// TIA Portal V15.1 export
// export: Created 2020-12-11T18:23:40.5486827Z, ExportSetting WithDefaults, WithReadOnly, DisplayName Totally Integrated Automation Portal, DisplayVersion V15.1 Update 4, DisplayName TIA Portal Openness, DisplayVersion V15.1, DisplayName SINAMICS Startdrive Advanced, DisplayVersion V15.1 Update3, DisplayName SINAMICS Startdrive G110M, G120, G120C, G120D, G120P, DisplayVersion V15.1 Update3, DisplayName SINAMICS Startdrive G130, G150, S120, S150, SINAMICS MV, S210, DisplayVersion V15.1 Update3, DisplayName STEP 7 Professional, DisplayVersion V15.1 Update 4, DisplayName STEP 7 Safety, DisplayVersion V15.1, DisplayName WinCC Professional, DisplayVersion V15.1 Update 4
PlcWatchTable "IO_ST_A"
  PlcTableCommentEntry   Comment="D1"
  PlcWatchTableEntry "Hello world"  Address=%I2001.0, DisplayFormat=Bool, ModifyTrigger=Permanent, MonitorTrigger=Permanent
  PlcWatchTableEntry ""SQ86/BA""  Address=%I2000.1, DisplayFormat=Bool, ModifyTrigger=Permanent, MonitorTrigger=Permanent
  PlcWatchTableEntry ""SQ87/BA""  Address=%I2001.1, DisplayFormat=Bool, ModifyTrigger=Permanent, MonitorTrigger=Permanent
  PlcWatchTableEntry ""SQ57/BA""  Address=%I2000.2, DisplayFormat=Bool, ModifyTrigger=Permanent, MonitorTrigger=Permanent
  PlcWatchTableEntry ""SQ58/BA""  Address=%I2001.2, DisplayFormat=Bool, ModifyTrigger=Permanent, MonitorTrigger=Permanent
  PlcWatchTableEntry ""SQ59/BA""  Address=%I2000.3, DisplayFormat=Bool, ModifyTrigger=Permanent, MonitorTrigger=Permanent
  PlcWatchTableEntry ""SQ60/BA""  Address=%I2001.3, DisplayFormat=Bool, ModifyTrigger=Permanent, MonitorTrigger=Permanent
  PlcWatchTableEntry ""SQ73/BA""  Address=%I2000.4, DisplayFormat=Bool, ModifyTrigger=Permanent, MonitorTrigger=Permanent
  PlcWatchTableEntry ""SQ74/BA""  Address=%I2001.4, DisplayFormat=Bool, ModifyTrigger=Permanent, MonitorTrigger=Permanent
  PlcWatchTableEntry ""SQ31/BA""  Address=%I2000.5, DisplayFormat=Bool, ModifyTrigger=Permanent, MonitorTrigger=Permanent
  PlcWatchTableEntry ""SQ32/BA""  Address=%I2001.5, DisplayFormat=Bool, ModifyTrigger=Permanent, MonitorTrigger=Permanent
  PlcWatchTableEntry ""FTC2/BA""  Address=%I2000.6, DisplayFormat=Bool, ModifyTrigger=Permanent, MonitorTrigger=Permanent
  PlcWatchTableEntry ""SQ15/BA""  Address=%I2001.6, DisplayFormat=Bool, ModifyTrigger=Permanent, MonitorTrigger=Permanent
  PlcWatchTableEntry ""FTC1/BA""  Address=%I2000.7, DisplayFormat=Bool, ModifyTrigger=Permanent, MonitorTrigger=Permanent
  PlcWatchTableEntry ""FTC3/BA""  Address=%I2001.7, DisplayFormat=Bool, ModifyTrigger=Permanent, MonitorTrigger=Permanent
  PlcTableCommentEntry   Comment="D2"
  PlcWatchTableEntry ""SQ61/BA""  Address=%I2002.0, DisplayFormat=Bool, ModifyTrigger=Permanent, MonitorTrigger=Permanent
  PlcWatchTableEntry ""SQ62/BA""  Address=%I2003.0, DisplayFormat=Bool, ModifyTrigger=Permanent, MonitorTrigger=Permanent
  PlcWatchTableEntry ""SQ66/BA""  Address=%I2002.1, DisplayFormat=Bool, ModifyTrigger=Permanent, MonitorTrigger=Permanent
  PlcWatchTableEntry ""SQ67/BA""  Address=%I2003.1, DisplayFormat=Bool, ModifyTrigger=Permanent, MonitorTrigger=Permanent
  PlcWatchTableEntry ""SQ68/BA""  Address=%I2002.2, DisplayFormat=Bool, ModifyTrigger=Permanent, MonitorTrigger=Permanent
  PlcWatchTableEntry ""SQ72/BA""  Address=%I2003.2, DisplayFormat=Bool, ModifyTrigger=Permanent, MonitorTrigger=Permanent
  PlcWatchTableEntry ""SQ8/BA""  Address=%I2002.3, DisplayFormat=Bool, ModifyTrigger=Permanent, MonitorTrigger=Permanent
  PlcWatchTableEntry ""SQ9/BA""  Address=%I2003.3, DisplayFormat=Bool, ModifyTrigger=Permanent, MonitorTrigger=Permanent
  PlcWatchTableEntry ""SQ80/BA""  Address=%I2002.4, DisplayFormat=Bool, ModifyTrigger=Permanent, MonitorTrigger=Permanent
  PlcWatchTableEntry ""SQ81/BA""  Address=%I2003.4, DisplayFormat=Bool, ModifyTrigger=Permanent, MonitorTrigger=Permanent
  PlcWatchTableEntry ""FTC15/BA""  Address=%I2002.5, DisplayFormat=Bool, ModifyTrigger=Permanent, MonitorTrigger=Permanent
  PlcWatchTableEntry ""FTC92/BA""  Address=%I2003.5, DisplayFormat=Bool, ModifyTrigger=Permanent, MonitorTrigger=Permanent
  PlcWatchTableEntry ""FTC93/BA""  Address=%I2002.6, DisplayFormat=Bool, ModifyTrigger=Permanent, MonitorTrigger=Permanent
  PlcWatchTableEntry ""FTC94/BA""  Address=%I2003.6, DisplayFormat=Bool, ModifyTrigger=Permanent, MonitorTrigger=Permanent
  PlcWatchTableEntry ""SQ_SPARE_31/BA""  Address=%I2002.7, DisplayFormat=Bool, ModifyTrigger=Permanent, MonitorTrigger=Permanent
  PlcWatchTableEntry ""SQ_SPARE_32/BA""  Address=%I2003.7, DisplayFormat=Bool, ModifyTrigger=Permanent, MonitorTrigger=Permanent
  PlcTableCommentEntry   Comment="D3 - REMOVED"
  PlcWatchTableEntry ""SQ_SPARE_33/BA""  Address=%I2004.0, DisplayFormat=Bool, ModifyTrigger=Permanent, MonitorTrigger=Permanent
  PlcWatchTableEntry ""SQ_SPARE_34/BA""  Address=%I2005.0, DisplayFormat=Bool, ModifyTrigger=Permanent, MonitorTrigger=Permanent
  PlcWatchTableEntry ""SQ_SPARE_35/BA""  Address=%I2004.1, DisplayFormat=Bool, ModifyTrigger=Permanent, MonitorTrigger=Permanent
  PlcWatchTableEntry ""SQ_SPARE_36/BA""  Address=%I2005.1, DisplayFormat=Bool, ModifyTrigger=Permanent, MonitorTrigger=Permanent
  PlcWatchTableEntry ""SQ_SPARE_37/BA""  Address=%I2004.2, DisplayFormat=Bool, ModifyTrigger=Permanent, MonitorTrigger=Permanent
  PlcWatchTableEntry ""SQ_SPARE_38/BA""  Address=%I2005.2, DisplayFormat=Bool, ModifyTrigger=Permanent, MonitorTrigger=Permanent
  PlcWatchTableEntry ""SQ_SPARE_39/BA""  Address=%I2004.3, DisplayFormat=Bool, ModifyTrigger=Permanent, MonitorTrigger=Permanent
  PlcWatchTableEntry ""SQ_SPARE_40/BA""  Address=%I2005.3, DisplayFormat=Bool, ModifyTrigger=Permanent, MonitorTrigger=Permanent
  PlcWatchTableEntry ""SQ_SPARE_41/BA""  Address=%I2004.4, DisplayFormat=Bool, ModifyTrigger=Permanent, MonitorTrigger=Permanent
  PlcWatchTableEntry ""SQ_SPARE_42/BA""  Address=%I2005.4, DisplayFormat=Bool, ModifyTrigger=Permanent, MonitorTrigger=Permanent
  PlcWatchTableEntry ""SQ_SPARE_43/BA""  Address=%I2004.5, DisplayFormat=Bool, ModifyTrigger=Permanent, MonitorTrigger=Permanent
  PlcWatchTableEntry ""SQ_SPARE_44/BA""  Address=%I2005.5, DisplayFormat=Bool, ModifyTrigger=Permanent, MonitorTrigger=Permanent
  PlcWatchTableEntry ""SQ_SPARE_45/BA""  Address=%I2004.6, DisplayFormat=Bool, ModifyTrigger=Permanent, MonitorTrigger=Permanent
  PlcWatchTableEntry ""SQ_SPARE_46/BA""  Address=%I2005.6, DisplayFormat=Bool, ModifyTrigger=Permanent, MonitorTrigger=Permanent
  PlcWatchTableEntry ""SQ_SPARE_47/BA""  Address=%I2004.7, DisplayFormat=Bool, ModifyTrigger=Permanent, MonitorTrigger=Permanent
  PlcWatchTableEntry ""SQ_SPARE_48/BA""  Address=%I2005.7, DisplayFormat=Bool, ModifyTrigger=Permanent, MonitorTrigger=Permanent
  PlcTableCommentEntry   Comment="D2A"
  PlcWatchTableEntry ""FTC5/BA""  Address=%I2006.0, DisplayFormat=Bool, ModifyTrigger=Permanent, MonitorTrigger=Permanent
  PlcWatchTableEntry ""FTC6/BA""  Address=%I2007.0, DisplayFormat=Bool, ModifyTrigger=Permanent, MonitorTrigger=Permanent
  PlcWatchTableEntry ""FTC7/BA""  Address=%I2006.1, DisplayFormat=Bool, ModifyTrigger=Permanent, MonitorTrigger=Permanent
  PlcWatchTableEntry ""SQ95/BA""  Address=%I2007.1, DisplayFormat=Bool, ModifyTrigger=Permanent, MonitorTrigger=Permanent
  PlcWatchTableEntry ""SQ_SPARE_99/BA""  Address=%I2006.2, DisplayFormat=Bool, ModifyTrigger=Permanent, MonitorTrigger=Permanent
  PlcWatchTableEntry ""SQ_SPARE_107/BA""  Address=%I2007.2, DisplayFormat=Bool, ModifyTrigger=Permanent, MonitorTrigger=Permanent
  PlcWatchTableEntry ""FTC90/BA""  Address=%I2006.3, DisplayFormat=Bool, ModifyTrigger=Permanent, MonitorTrigger=Permanent
  PlcWatchTableEntry ""SQ96/BA""  Address=%I2007.3, DisplayFormat=Bool, ModifyTrigger=Permanent, MonitorTrigger=Permanent
  PlcWatchTableEntry ""SQ_SPARE_101/BA""  Address=%I2006.4, DisplayFormat=Bool, ModifyTrigger=Permanent, MonitorTrigger=Permanent
  PlcWatchTableEntry ""SQ_SPARE_109/BA""  Address=%I2007.4, DisplayFormat=Bool, ModifyTrigger=Permanent, MonitorTrigger=Permanent
  PlcWatchTableEntry ""SQ_SPARE_102/BA""  Address=%I2006.5, DisplayFormat=Bool, ModifyTrigger=Permanent, MonitorTrigger=Permanent
  PlcWatchTableEntry ""SQ_SPARE_110/BA""  Address=%I2007.5, DisplayFormat=Bool, ModifyTrigger=Permanent, MonitorTrigger=Permanent
  PlcWatchTableEntry ""SQ_SPARE_103/BA""  Address=%I2006.6, DisplayFormat=Bool, ModifyTrigger=Permanent, MonitorTrigger=Permanent
  PlcWatchTableEntry ""SQ_SPARE_111/BA""  Address=%I2007.6, DisplayFormat=Bool, ModifyTrigger=Permanent, MonitorTrigger=Permanent
  PlcWatchTableEntry ""SQ_SPARE_104/BA""  Address=%I2006.7, DisplayFormat=Bool, ModifyTrigger=Permanent, MonitorTrigger=Permanent
  PlcWatchTableEntry ""SQ_SPARE_112/BA""  Address=%I2007.7, DisplayFormat=Bool, ModifyTrigger=Permanent, MonitorTrigger=Permanent
  PlcTableCommentEntry   Comment="D4"
  PlcWatchTableEntry ""SQ44/BA""  Address=%I2100.0, DisplayFormat=Bool, ModifyTrigger=Permanent, MonitorTrigger=Permanent
  PlcWatchTableEntry ""SQ45/BA""  Address=%I2101.0, DisplayFormat=Bool, ModifyTrigger=Permanent, MonitorTrigger=Permanent
  PlcWatchTableEntry ""SQ89/BA""  Address=%I2101.1, DisplayFormat=Bool, ModifyTrigger=Permanent, MonitorTrigger=Permanent
  PlcWatchTableEntry ""SQ88/BA""  Address=%I2100.1, DisplayFormat=Bool, ModifyTrigger=Permanent, MonitorTrigger=Permanent
  PlcWatchTableEntry ""SQ48/BA""  Address=%I2100.2, DisplayFormat=Bool, ModifyTrigger=Permanent, MonitorTrigger=Permanent
  PlcWatchTableEntry ""SQ49/BA""  Address=%I2101.2, DisplayFormat=Bool, ModifyTrigger=Permanent, MonitorTrigger=Permanent
  PlcWatchTableEntry ""SQ50/BA""  Address=%I2100.3, DisplayFormat=Bool, ModifyTrigger=Permanent, MonitorTrigger=Permanent
  PlcWatchTableEntry ""SQ51/BA""  Address=%I2101.3, DisplayFormat=Bool, ModifyTrigger=Permanent, MonitorTrigger=Permanent
  PlcWatchTableEntry ""SQ75/BA""  Address=%I2100.4, DisplayFormat=Bool, ModifyTrigger=Permanent, MonitorTrigger=Permanent
  PlcWatchTableEntry ""SQ76/BA""  Address=%I2101.4, DisplayFormat=Bool, ModifyTrigger=Permanent, MonitorTrigger=Permanent
  PlcWatchTableEntry ""SQ18/BA""  Address=%I2100.5, DisplayFormat=Bool, ModifyTrigger=Permanent, MonitorTrigger=Permanent
  PlcWatchTableEntry ""SQ19/BA""  Address=%I2101.5, DisplayFormat=Bool, ModifyTrigger=Permanent, MonitorTrigger=Permanent
  PlcWatchTableEntry ""SQ97/BA""  Address=%I2100.6, DisplayFormat=Bool, ModifyTrigger=Permanent, MonitorTrigger=Permanent
  PlcWatchTableEntry ""SQ17/BA""  Address=%I2101.6, DisplayFormat=Bool, ModifyTrigger=Permanent, MonitorTrigger=Permanent
  PlcWatchTableEntry ""SQ98/BA""  Address=%I2100.7, DisplayFormat=Bool, ModifyTrigger=Permanent, MonitorTrigger=Permanent
  PlcWatchTableEntry ""SQ_SPARE_64/BA""  Address=%I2101.7, DisplayFormat=Bool, ModifyTrigger=Permanent, MonitorTrigger=Permanent
  PlcTableCommentEntry   Comment="D5 - REMOVED"
  PlcWatchTableEntry ""SQ_SPARE_65/BA""  Address=%I2102.0, DisplayFormat=Bool, ModifyTrigger=Permanent, MonitorTrigger=Permanent
  PlcWatchTableEntry ""SQ_SPARE_66/BA""  Address=%I2103.0, DisplayFormat=Bool, ModifyTrigger=Permanent, MonitorTrigger=Permanent
  PlcWatchTableEntry ""SQ_SPARE_67/BA""  Address=%I2102.1, DisplayFormat=Bool, ModifyTrigger=Permanent, MonitorTrigger=Permanent
  PlcWatchTableEntry ""SQ_SPARE_68/BA""  Address=%I2103.1, DisplayFormat=Bool, ModifyTrigger=Permanent, MonitorTrigger=Permanent
  PlcWatchTableEntry ""SQ_SPARE_69/BA""  Address=%I2102.2, DisplayFormat=Bool, ModifyTrigger=Permanent, MonitorTrigger=Permanent
  PlcWatchTableEntry ""SQ_SPARE_70/BA""  Address=%I2103.2, DisplayFormat=Bool, ModifyTrigger=Permanent, MonitorTrigger=Permanent
  PlcWatchTableEntry ""SQ_SPARE_71/BA""  Address=%I2102.3, DisplayFormat=Bool, ModifyTrigger=Permanent, MonitorTrigger=Permanent
  PlcWatchTableEntry ""SQ_SPARE_72/BA""  Address=%I2103.3, DisplayFormat=Bool, ModifyTrigger=Permanent, MonitorTrigger=Permanent
  PlcWatchTableEntry ""SQ_SPARE_73/BA""  Address=%I2102.4, DisplayFormat=Bool, ModifyTrigger=Permanent, MonitorTrigger=Permanent
  PlcWatchTableEntry ""SQ_SPARE_74/BA""  Address=%I2103.4, DisplayFormat=Bool, ModifyTrigger=Permanent, MonitorTrigger=Permanent
  PlcWatchTableEntry ""SQ_SPARE_75/BA""  Address=%I2102.5, DisplayFormat=Bool, ModifyTrigger=Permanent, MonitorTrigger=Permanent
  PlcWatchTableEntry ""SQ_SPARE_76/BA""  Address=%I2103.5, DisplayFormat=Bool, ModifyTrigger=Permanent, MonitorTrigger=Permanent
  PlcWatchTableEntry ""SQ_SPARE_77/BA""  Address=%I2102.6, DisplayFormat=Bool, ModifyTrigger=Permanent, MonitorTrigger=Permanent
  PlcWatchTableEntry ""SQ_SPARE_78/BA""  Address=%I2103.6, DisplayFormat=Bool, ModifyTrigger=Permanent, MonitorTrigger=Permanent
  PlcWatchTableEntry ""SQ_SPARE_79/BA""  Address=%I2102.7, DisplayFormat=Bool, ModifyTrigger=Permanent, MonitorTrigger=Permanent
  PlcWatchTableEntry ""SQ_SPARE_80/BA""  Address=%I2103.7, DisplayFormat=Bool, ModifyTrigger=Permanent, MonitorTrigger=Permanent
  PlcTableCommentEntry   Comment="D6"
  PlcWatchTableEntry ""SQ69/BA""  Address=%I2104.0, DisplayFormat=Bool, ModifyTrigger=Permanent, MonitorTrigger=Permanent
  PlcWatchTableEntry ""SQ70/BA""  Address=%I2105.0, DisplayFormat=Bool, ModifyTrigger=Permanent, MonitorTrigger=Permanent
  PlcWatchTableEntry ""SQ71/BA""  Address=%I2104.1, DisplayFormat=Bool, ModifyTrigger=Permanent, MonitorTrigger=Permanent
  PlcWatchTableEntry ""SQ77/BA""  Address=%I2105.1, DisplayFormat=Bool, ModifyTrigger=Permanent, MonitorTrigger=Permanent
  PlcWatchTableEntry ""SQ78/BA""  Address=%I2104.2, DisplayFormat=Bool, ModifyTrigger=Permanent, MonitorTrigger=Permanent
  PlcWatchTableEntry ""SQ79/BA""  Address=%I2105.2, DisplayFormat=Bool, ModifyTrigger=Permanent, MonitorTrigger=Permanent
  PlcWatchTableEntry ""SQ6/BA""  Address=%I2104.3, DisplayFormat=Bool, ModifyTrigger=Permanent, MonitorTrigger=Permanent
  PlcWatchTableEntry ""SQ7/BA""  Address=%I2105.3, DisplayFormat=Bool, ModifyTrigger=Permanent, MonitorTrigger=Permanent
  PlcWatchTableEntry ""SQ82/BA""  Address=%I2104.4, DisplayFormat=Bool, ModifyTrigger=Permanent, MonitorTrigger=Permanent
  PlcWatchTableEntry ""SQ83/BA""  Address=%I2105.4, DisplayFormat=Bool, ModifyTrigger=Permanent, MonitorTrigger=Permanent
  PlcWatchTableEntry ""SQ_SPARE_91/BA""  Address=%I2104.5, DisplayFormat=Bool, ModifyTrigger=Permanent, MonitorTrigger=Permanent
  PlcWatchTableEntry ""SQ_SPARE_92/BA""  Address=%I2105.5, DisplayFormat=Bool, ModifyTrigger=Permanent, MonitorTrigger=Permanent
  PlcWatchTableEntry ""SQ_SPARE_93/BA""  Address=%I2104.6, DisplayFormat=Bool, ModifyTrigger=Permanent, MonitorTrigger=Permanent
  PlcWatchTableEntry ""SQ_SPARE_94/BA""  Address=%I2105.6, DisplayFormat=Bool, ModifyTrigger=Permanent, MonitorTrigger=Permanent
  PlcWatchTableEntry ""SQ_SPARE_95/BA""  Address=%I2104.7, DisplayFormat=Bool, ModifyTrigger=Permanent, MonitorTrigger=Permanent
  PlcWatchTableEntry ""SQ_SPARE_96/BA""  Address=%I2105.7, DisplayFormat=Bool, ModifyTrigger=Permanent, MonitorTrigger=Permanent
  PlcTableCommentEntry   Comment="D6A"
  PlcWatchTableEntry ""SQ_SPARE_113/BA""  Address=%I2106.0, DisplayFormat=Bool, ModifyTrigger=Permanent, MonitorTrigger=Permanent
  PlcWatchTableEntry ""SQ_SPARE_114/BA""  Address=%I2106.1, DisplayFormat=Bool, ModifyTrigger=Permanent, MonitorTrigger=Permanent
  PlcWatchTableEntry ""SQ_SPARE_115/BA""  Address=%I2106.2, DisplayFormat=Bool, ModifyTrigger=Permanent, MonitorTrigger=Permanent
  PlcWatchTableEntry ""SQ_SPARE_116/BA""  Address=%I2106.3, DisplayFormat=Bool, ModifyTrigger=Permanent, MonitorTrigger=Permanent
  PlcWatchTableEntry ""FTC91/BA""  Address=%I2106.4, DisplayFormat=Bool, ModifyTrigger=Permanent, MonitorTrigger=Permanent
  PlcWatchTableEntry ""SQ_SPARE_118/BA""  Address=%I2106.5, DisplayFormat=Bool, ModifyTrigger=Permanent, MonitorTrigger=Permanent
  PlcWatchTableEntry ""SQ_SPARE_119/BA""  Address=%I2106.6, DisplayFormat=Bool, ModifyTrigger=Permanent, MonitorTrigger=Permanent
  PlcWatchTableEntry ""SQ_SPARE_120/BA""  Address=%I2106.7, DisplayFormat=Bool, ModifyTrigger=Permanent, MonitorTrigger=Permanent
  PlcWatchTableEntry ""SQ_SPARE_121/BA""  Address=%I2107.0, DisplayFormat=Bool, ModifyTrigger=Permanent, MonitorTrigger=Permanent
  PlcWatchTableEntry ""SQ_SPARE_122/BA""  Address=%I2107.1, DisplayFormat=Bool, ModifyTrigger=Permanent, MonitorTrigger=Permanent
  PlcWatchTableEntry ""SQ_SPARE_123/BA""  Address=%I2107.2, DisplayFormat=Bool, ModifyTrigger=Permanent, MonitorTrigger=Permanent
  PlcWatchTableEntry ""SQ_SPARE_124/BA""  Address=%I2107.3, DisplayFormat=Bool, ModifyTrigger=Permanent, MonitorTrigger=Permanent
  PlcWatchTableEntry ""SQ_SPARE_125/BA""  Address=%I2107.4, DisplayFormat=Bool, ModifyTrigger=Permanent, MonitorTrigger=Permanent
  PlcWatchTableEntry ""SQ_SPARE_126/BA""  Address=%I2107.5, DisplayFormat=Bool, ModifyTrigger=Permanent, MonitorTrigger=Permanent
  PlcWatchTableEntry ""SQ_SPARE_127/BA""  Address=%I2107.6, DisplayFormat=Bool, ModifyTrigger=Permanent, MonitorTrigger=Permanent
  PlcWatchTableEntry ""SQ_SPARE_128/BA""  Address=%I2107.7, DisplayFormat=Bool, ModifyTrigger=Permanent, MonitorTrigger=Permanent
  PlcWatchTableEntry   DisplayFormat=Undef, ModifyTrigger=Undef, MonitorTrigger=Undef
  PlcWatchTableEntry   DisplayFormat=Undef, ModifyTrigger=Undef, MonitorTrigger=Undef
  PlcWatchTableEntry   DisplayFormat=Undef, ModifyTrigger=Undef, MonitorTrigger=Undef
  PlcWatchTableEntry   DisplayFormat=Undef, ModifyTrigger=Undef, MonitorTrigger=Undef
  PlcWatchTableEntry   Address=%QB0, DisplayFormat=Hex, ModifyTrigger=Permanent, ModifyValue=16#FF, MonitorTrigger=Permanent
  PlcWatchTableEntry ""Y1A/BA""  Address=%Q2000.0, DisplayFormat=Bool, ModifyTrigger=Permanent, MonitorTrigger=Permanent
  PlcWatchTableEntry ""Y1B/BA""  Address=%Q2000.1, DisplayFormat=Bool, ModifyTrigger=Permanent, MonitorTrigger=Permanent
  PlcWatchTableEntry ""Y2A/BA""  Address=%Q2000.2, DisplayFormat=Bool, ModifyTrigger=Permanent, MonitorTrigger=Permanent
  PlcWatchTableEntry ""Y2B/BA""  Address=%Q2000.3, DisplayFormat=Bool, ModifyTrigger=Permanent, MonitorTrigger=Permanent
  PlcWatchTableEntry ""Y3A/BA""  Address=%Q2000.4, DisplayFormat=Bool, ModifyTrigger=Permanent, MonitorTrigger=Permanent
  PlcWatchTableEntry ""Y3B/BA""  Address=%Q2000.5, DisplayFormat=Bool, ModifyTrigger=Permanent, MonitorTrigger=Permanent
  PlcWatchTableEntry ""Y4A/BA""  Address=%Q2000.6, DisplayFormat=Bool, ModifyTrigger=Permanent, MonitorTrigger=Permanent
  PlcWatchTableEntry ""Y4B/BA""  Address=%Q2000.7, DisplayFormat=Bool, ModifyTrigger=Permanent, MonitorTrigger=Permanent
  PlcWatchTableEntry ""Y5A/BA""  Address=%Q2001.0, DisplayFormat=Bool, ModifyTrigger=Permanent, MonitorTrigger=Permanent
  PlcWatchTableEntry ""Y5B/BA""  Address=%Q2001.1, DisplayFormat=Bool, ModifyTrigger=Permanent, MonitorTrigger=Permanent
  PlcWatchTableEntry ""Y6A/BA""  Address=%Q2001.2, DisplayFormat=Bool, ModifyTrigger=Permanent, MonitorTrigger=Permanent
  PlcWatchTableEntry ""Y6B/BA""  Address=%Q2001.3, DisplayFormat=Bool, ModifyTrigger=Permanent, MonitorTrigger=Permanent
  PlcWatchTableEntry ""Y7A/BA""  Address=%Q2001.4, DisplayFormat=Bool, ModifyTrigger=Permanent, MonitorTrigger=Permanent
  PlcWatchTableEntry ""Y7B/BA""  Address=%Q2001.5, DisplayFormat=Bool, ModifyTrigger=Permanent, MonitorTrigger=Permanent
  PlcWatchTableEntry ""Y8A/BA""  Address=%Q2001.6, DisplayFormat=Bool, ModifyTrigger=Permanent, MonitorTrigger=Permanent
  PlcWatchTableEntry ""Y8B/BA""  Address=%Q2001.7, DisplayFormat=Bool, ModifyTrigger=Permanent, MonitorTrigger=Permanent
  PlcWatchTableEntry ""Y9A/BA""  Address=%Q2002.0, DisplayFormat=Bool, ModifyTrigger=Permanent, MonitorTrigger=Permanent
  PlcWatchTableEntry ""Y9B/BA""  Address=%Q2002.1, DisplayFormat=Bool, ModifyTrigger=Permanent, MonitorTrigger=Permanent
  PlcWatchTableEntry ""Y10A/BA""  Address=%Q2002.2, DisplayFormat=Bool, ModifyTrigger=Permanent, MonitorTrigger=Permanent
  PlcWatchTableEntry ""Y10B/BA""  Address=%Q2002.3, DisplayFormat=Bool, ModifyTrigger=Permanent, MonitorTrigger=Permanent
  PlcWatchTableEntry ""Y11A/BA""  Address=%Q2002.4, DisplayFormat=Bool, ModifyTrigger=Permanent, MonitorTrigger=Permanent
  PlcWatchTableEntry ""Y11B/BA""  Address=%Q2002.5, DisplayFormat=Bool, ModifyTrigger=Permanent, MonitorTrigger=Permanent
  PlcWatchTableEntry ""Y12A/BA""  Address=%Q2002.6, DisplayFormat=Bool, ModifyTrigger=Permanent, MonitorTrigger=Permanent
  PlcWatchTableEntry ""Y12B/BA""  Address=%Q2002.7, DisplayFormat=Bool, ModifyTrigger=Permanent, MonitorTrigger=Permanent
  PlcWatchTableEntry ""Y13A/BA""  Address=%Q2003.0, DisplayFormat=Bool, ModifyTrigger=Permanent, MonitorTrigger=Permanent
  PlcWatchTableEntry ""Y13B/BA""  Address=%Q2003.1, DisplayFormat=Bool, ModifyTrigger=Permanent, MonitorTrigger=Permanent
  PlcWatchTableEntry ""Y14A/BA""  Address=%Q2003.2, DisplayFormat=Bool, ModifyTrigger=Permanent, MonitorTrigger=Permanent
  PlcWatchTableEntry ""Y14B/BA""  Address=%Q2003.3, DisplayFormat=Bool, ModifyTrigger=Permanent, MonitorTrigger=Permanent
  PlcWatchTableEntry ""Y15A/BA""  Address=%Q2003.4, DisplayFormat=Bool, ModifyTrigger=Permanent, MonitorTrigger=Permanent
  PlcWatchTableEntry ""EV_SPARE_30/BA""  Address=%Q2003.5, DisplayFormat=Bool, ModifyTrigger=Permanent, MonitorTrigger=Permanent
  PlcWatchTableEntry ""EV_SPARE_31/BA""  Address=%Q2003.6, DisplayFormat=Bool, ModifyTrigger=Permanent, MonitorTrigger=Permanent
  PlcWatchTableEntry ""EV_SPARE_32/BA""  Address=%Q2003.7, DisplayFormat=Bool, ModifyTrigger=Permanent, MonitorTrigger=Permanent
  PlcWatchTableEntry ""Y17A/BA""  Address=%Q2100.0, DisplayFormat=Bool, ModifyTrigger=Permanent, MonitorTrigger=Permanent
  PlcWatchTableEntry ""Y17B/BA""  Address=%Q2100.1, DisplayFormat=Bool, ModifyTrigger=Permanent, MonitorTrigger=Permanent
  PlcWatchTableEntry ""Y18A/BA""  Address=%Q2100.2, DisplayFormat=Bool, ModifyTrigger=Permanent, MonitorTrigger=Permanent
  PlcWatchTableEntry ""Y18B/BA""  Address=%Q2100.3, DisplayFormat=Bool, ModifyTrigger=Permanent, MonitorTrigger=Permanent
  PlcWatchTableEntry ""Y19A/BA""  Address=%Q2100.4, DisplayFormat=Bool, ModifyTrigger=Permanent, MonitorTrigger=Permanent
  PlcWatchTableEntry ""Y19B/BA""  Address=%Q2100.5, DisplayFormat=Bool, ModifyTrigger=Permanent, MonitorTrigger=Permanent
  PlcWatchTableEntry ""Y20A/BA""  Address=%Q2100.6, DisplayFormat=Bool, ModifyTrigger=Permanent, MonitorTrigger=Permanent
  PlcWatchTableEntry ""Y20B/BA""  Address=%Q2100.7, DisplayFormat=Bool, ModifyTrigger=Permanent, MonitorTrigger=Permanent
  PlcWatchTableEntry ""Y21A/BA""  Address=%Q2101.0, DisplayFormat=Bool, ModifyTrigger=Permanent, MonitorTrigger=Permanent
  PlcWatchTableEntry ""Y21B/BA""  Address=%Q2101.1, DisplayFormat=Bool, ModifyTrigger=Permanent, MonitorTrigger=Permanent
  PlcWatchTableEntry ""Y22A/BA""  Address=%Q2101.2, DisplayFormat=Bool, ModifyTrigger=Permanent, MonitorTrigger=Permanent
  PlcWatchTableEntry ""Y22B/BA""  Address=%Q2101.3, DisplayFormat=Bool, ModifyTrigger=Permanent, MonitorTrigger=Permanent
  PlcWatchTableEntry ""Y23A/BA""  Address=%Q2101.4, DisplayFormat=Bool, ModifyTrigger=Permanent, MonitorTrigger=Permanent
  PlcWatchTableEntry ""Y23B/BA""  Address=%Q2101.5, DisplayFormat=Bool, ModifyTrigger=Permanent, MonitorTrigger=Permanent
  PlcWatchTableEntry ""Y24A/BA""  Address=%Q2101.6, DisplayFormat=Bool, ModifyTrigger=Permanent, MonitorTrigger=Permanent
  PlcWatchTableEntry ""Y24B/BA""  Address=%Q2101.7, DisplayFormat=Bool, ModifyTrigger=Permanent, MonitorTrigger=Permanent
  PlcWatchTableEntry ""Y25A/BA""  Address=%Q2102.0, DisplayFormat=Bool, ModifyTrigger=Permanent, MonitorTrigger=Permanent
  PlcWatchTableEntry ""Y25B/BA""  Address=%Q2102.1, DisplayFormat=Bool, ModifyTrigger=Permanent, MonitorTrigger=Permanent
  PlcWatchTableEntry ""Y26A/BA""  Address=%Q2102.2, DisplayFormat=Bool, ModifyTrigger=Permanent, MonitorTrigger=Permanent
  PlcWatchTableEntry ""Y26B/BA""  Address=%Q2102.3, DisplayFormat=Bool, ModifyTrigger=Permanent, MonitorTrigger=Permanent
  PlcWatchTableEntry ""Y27A/BA""  Address=%Q2102.4, DisplayFormat=Bool, ModifyTrigger=Permanent, MonitorTrigger=Permanent
  PlcWatchTableEntry ""Y27B/BA""  Address=%Q2102.5, DisplayFormat=Bool, ModifyTrigger=Permanent, MonitorTrigger=Permanent
  PlcWatchTableEntry ""Y28A/BA""  Address=%Q2102.6, DisplayFormat=Bool, ModifyTrigger=Permanent, MonitorTrigger=Permanent
  PlcWatchTableEntry ""Y28B/BA""  Address=%Q2102.7, DisplayFormat=Bool, ModifyTrigger=Permanent, MonitorTrigger=Permanent
  PlcWatchTableEntry ""Y29A/BA""  Address=%Q2103.0, DisplayFormat=Bool, ModifyTrigger=Permanent, MonitorTrigger=Permanent
  PlcWatchTableEntry ""EV_SPARE_58/BA""  Address=%Q2103.1, DisplayFormat=Bool, ModifyTrigger=Permanent, MonitorTrigger=Permanent
  PlcWatchTableEntry ""EV_SPARE_59/BA""  Address=%Q2103.2, DisplayFormat=Bool, ModifyTrigger=Permanent, MonitorTrigger=Permanent
  PlcWatchTableEntry ""EV_SPARE_60/BA""  Address=%Q2103.3, DisplayFormat=Bool, ModifyTrigger=Permanent, MonitorTrigger=Permanent
  PlcWatchTableEntry ""EV_SPARE_61/BA""  Address=%Q2103.4, DisplayFormat=Bool, ModifyTrigger=Permanent, MonitorTrigger=Permanent
  PlcWatchTableEntry ""EV_SPARE_62/BA""  Address=%Q2103.5, DisplayFormat=Bool, ModifyTrigger=Permanent, MonitorTrigger=Permanent
  PlcWatchTableEntry ""EV_SPARE_63/BA""  Address=%Q2103.6, DisplayFormat=Bool, ModifyTrigger=Permanent, MonitorTrigger=Permanent
  PlcWatchTableEntry ""EV_SPARE_64/BA""  Address=%Q2103.7, DisplayFormat=Bool, ModifyTrigger=Permanent, MonitorTrigger=Permanent
  PlcWatchTableEntry   Address=%Q2200.0, DisplayFormat=Bool, ModifyTrigger=Permanent, MonitorTrigger=Permanent
  PlcWatchTableEntry   Address=%Q2200.1, DisplayFormat=Bool, ModifyTrigger=Permanent, MonitorTrigger=Permanent
  PlcWatchTableEntry   Address=%Q2200.2, DisplayFormat=Bool, ModifyTrigger=Permanent, MonitorTrigger=Permanent
  PlcWatchTableEntry   Address=%Q2200.3, DisplayFormat=Bool, ModifyTrigger=Permanent, MonitorTrigger=Permanent
  PlcWatchTableEntry   Address=%Q2200.4, DisplayFormat=Bool, ModifyTrigger=Permanent, MonitorTrigger=Permanent
  PlcWatchTableEntry   Address=%Q2200.5, DisplayFormat=Bool, ModifyTrigger=Permanent, MonitorTrigger=Permanent
  PlcWatchTableEntry   Address=%Q2200.6, DisplayFormat=Bool, ModifyTrigger=Permanent, MonitorTrigger=Permanent
  PlcWatchTableEntry   Address=%Q2200.7, DisplayFormat=Bool, ModifyTrigger=Permanent, MonitorTrigger=Permanent
  PlcWatchTableEntry   Address=%Q2201.0, DisplayFormat=Bool, ModifyTrigger=Permanent, MonitorTrigger=Permanent
  PlcWatchTableEntry   Address=%Q2201.1, DisplayFormat=Bool, ModifyTrigger=Permanent, MonitorTrigger=Permanent
  PlcWatchTableEntry   Address=%Q2201.2, DisplayFormat=Bool, ModifyTrigger=Permanent, MonitorTrigger=Permanent
  PlcWatchTableEntry   Address=%Q2201.3, DisplayFormat=Bool, ModifyTrigger=Permanent, MonitorTrigger=Permanent
  PlcWatchTableEntry   Address=%Q2201.4, DisplayFormat=Bool, ModifyTrigger=Permanent, MonitorTrigger=Permanent
  PlcWatchTableEntry   Address=%Q2201.5, DisplayFormat=Bool, ModifyTrigger=Permanent, MonitorTrigger=Permanent
  PlcWatchTableEntry   Address=%Q2201.6, DisplayFormat=Bool, ModifyTrigger=Permanent, MonitorTrigger=Permanent
  PlcWatchTableEntry   Address=%Q2201.7, DisplayFormat=Bool, ModifyTrigger=Permanent, MonitorTrigger=Permanent
  PlcWatchTableEntry   Address=%Q2202.0, DisplayFormat=Bool, ModifyTrigger=Permanent, MonitorTrigger=Permanent
  PlcWatchTableEntry   Address=%Q2202.1, DisplayFormat=Bool, ModifyTrigger=Permanent, MonitorTrigger=Permanent
  PlcWatchTableEntry   Address=%Q2202.2, DisplayFormat=Bool, ModifyTrigger=Permanent, MonitorTrigger=Permanent
  PlcWatchTableEntry   Address=%Q2202.3, DisplayFormat=Bool, ModifyTrigger=Permanent, MonitorTrigger=Permanent
  PlcWatchTableEntry   Address=%Q2202.4, DisplayFormat=Bool, ModifyTrigger=Permanent, MonitorTrigger=Permanent
  PlcWatchTableEntry   Address=%Q2202.5, DisplayFormat=Bool, ModifyTrigger=Permanent, MonitorTrigger=Permanent
  PlcWatchTableEntry   Address=%Q2202.6, DisplayFormat=Bool, ModifyTrigger=Permanent, MonitorTrigger=Permanent
  PlcWatchTableEntry   Address=%Q2202.7, DisplayFormat=Bool, ModifyTrigger=Permanent, MonitorTrigger=Permanent
  PlcWatchTableEntry   Address=%Q2203.0, DisplayFormat=Bool, ModifyTrigger=Permanent, MonitorTrigger=Permanent
  PlcWatchTableEntry   Address=%Q2203.1, DisplayFormat=Bool, ModifyTrigger=Permanent, MonitorTrigger=Permanent
  PlcWatchTableEntry   Address=%Q2203.2, DisplayFormat=Bool, ModifyTrigger=Permanent, MonitorTrigger=Permanent
  PlcWatchTableEntry   Address=%Q2204.7, DisplayFormat=Bool, ModifyTrigger=Permanent, MonitorTrigger=Permanent
  PlcWatchTableEntry   Address=%Q2204.6, DisplayFormat=Bool, ModifyTrigger=Permanent, MonitorTrigger=Permanent
  PlcWatchTableEntry   Address=%QW2220, DisplayFormat=DEC_signed, ModifyTrigger=Permanent, ModifyValue=32000, MonitorTrigger=Permanent
  PlcWatchTableEntry   DisplayFormat=Undef, ModifyTrigger=Undef, MonitorTrigger=Undef
  PlcWatchTableEntry   DisplayFormat=Undef, ModifyTrigger=Undef, MonitorTrigger=Undef
  PlcWatchTableEntry ""Y_GLUE_1A_SX/BA""  Address=%Q15.3, DisplayFormat=Bool, ModifyTrigger=Permanent, MonitorTrigger=Permanent
  PlcWatchTableEntry ""Y_GLUE_1B_SX/BA""  Address=%Q15.4, DisplayFormat=Bool, ModifyTrigger=Permanent, MonitorTrigger=Permanent
  PlcWatchTableEntry ""Y_GLUE_1A_DX/BA""  Address=%Q15.5, DisplayFormat=Bool, ModifyTrigger=Permanent, MonitorTrigger=Permanent
  PlcWatchTableEntry ""Y_GLUE_1B_DX/BA""  Address=%Q15.6, DisplayFormat=Bool, ModifyTrigger=Permanent, MonitorTrigger=Permanent
  PlcWatchTableEntry ""Y_GLUE_2A_SX/BA""  Address=%Q15.7, DisplayFormat=Bool, ModifyTrigger=Permanent, MonitorTrigger=Permanent
  PlcWatchTableEntry ""Y_GLUE_2A_DX/BA""  Address=%Q16.0, DisplayFormat=Bool, ModifyTrigger=Permanent, MonitorTrigger=Permanent
  PlcWatchTableEntry "Prova"  Address=M77.5, DisplayFormat=Bool, ModifyTrigger=Permanent, MonitorTrigger=Permanent
